(* PLC project Unnamed, Unknown Unnamed 1 *)
(* stored: creationDateTime 2023-03-10T10:37:17, modificationDateTime 2023-03-23T23:20:19 *)

(* SIEMENS AG- Beispielprogramm *)
FUNCTION_BLOCK Sports_Hall_Lighting
  VAR_INPUT
    IN1 : BOOL;
    IN2 : BOOL;
    IN3 : BOOL;
    IN4 : BOOL;
    TIME4 : BOOL;
    TIME9 : BOOL;
    TIME14 : BOOL;
    TIME18 : BOOL;
  END_VAR
  VAR_OUTPUT
    OUT1 : BOOL;
    OUT2 : BOOL;
    OUT3 : BOOL;
    OUT4 : BOOL;
  END_VAR
  VAR
    PT1m : TIME;
    RS0 : RS;
    RS1 : RS;
    RS2 : RS;
    TON0 : TON;
  END_VAR
  VAR  (* added by the conversion: wires and edge detectors of the diagram *)
    _OR2_OUT : BOOL;
    _OR1_OUT : BOOL;
  END_VAR

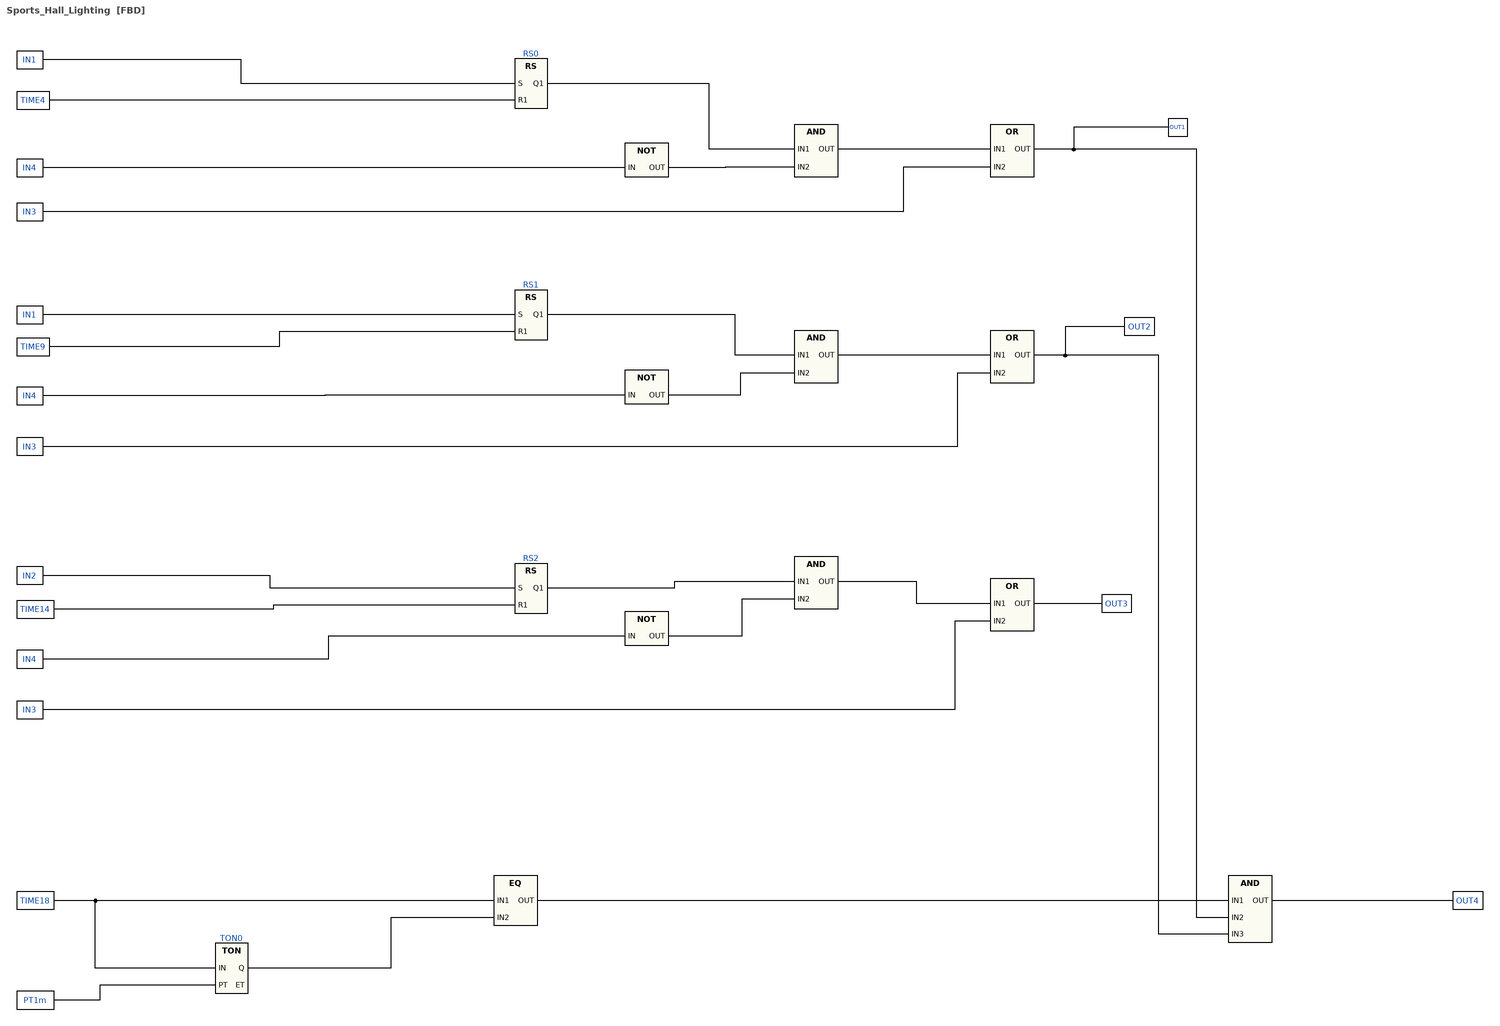
(* FBD diagram, written out as Structured Text *)
RS0(S := IN1, R1 := TIME4);
_OR2_OUT := RS0.Q1 AND NOT IN4 OR IN3;
OUT1 := _OR2_OUT;
RS1(S := IN1, R1 := TIME9);
_OR1_OUT := RS1.Q1 AND NOT IN4 OR IN3;
OUT2 := _OR1_OUT;
RS2(S := IN2, R1 := TIME14);
OUT3 := RS2.Q1 AND NOT IN4 OR IN3;
TON0(IN := TIME18, PT := PT1m);
OUT4 := TIME18 = TON0.Q AND _OR2_OUT AND _OR1_OUT;
END_FUNCTION_BLOCK

CONFIGURATION config
  RESOURCE resource1 ON PLC
  END_RESOURCE
END_CONFIGURATION
